PROGRAM P_Demo_BE32_TO_HOST
VAR
    bResult : DWORD; // BE32_TO_HOST 的返回值
    bRun    : BOOL; // 触发一次调用
END_VAR

// ============================================================
// Tc2_Utilities.BE32_TO_HOST 演示程序（FUNCTION）
// ============================================================
// 验证步骤：
//   1. 引用 Tc2_Utilities（及依赖类型所在的库）
//   2. 编译 + 登录
//   3. 强制 bRun := TRUE 一个周期
//   4. 观察 bResult 应为 16#12345678
// ============================================================

IF bRun THEN
    bResult := BE32_TO_HOST(16#78563412);
    bRun := FALSE;
END_IF;

END_PROGRAM

(* stored: Version 1.1.0.1, ProductVersion 3.1.4024.5
   POU P_Demo_BE32_TO_HOST: Id {cc01ed77-095c-5cc9-afa5-ee272ac53f49}, SpecialFunc None *)
